INTERFACE I_TempSensor

PROPERTY P_DegreesC : real
GET
END_GET
SET
END_SET
END_PROPERTY

PROPERTY P_DegreesF : real
GET
END_GET
END_PROPERTY

END_INTERFACE

(* stored: Version 1.1.0.1, ProductVersion 3.1.4022.12
   Itf I_TempSensor: Id {a3014177-8552-4fbc-b769-cfbd5546c312}
   Property P_DegreesC: Id {9731390f-d712-4ca9-89b0-b76b5a51722f}
   Get Get: Id {649236ed-2399-434c-9413-6554a9a9b4e9}
   Set Set: Id {b43a88e4-6f31-4150-a5ee-134f6ec71b78}
   Property P_DegreesF: Id {ac113eaa-529b-4dbe-b267-6677b9066c97}
   Get Get: Id {dbac1d45-0286-473e-977f-ce0f315bc18d} *)
